FUNCTION_BLOCK FB_SerialCom
VAR_IN_OUT
	RxBuffer	: ComBuffer;
	TxBuffer	: ComBuffer;
END_VAR

VAR
	fbSend		: SendString;
	bSendBusy	: BOOL;
	eSendErrorID: ComError_t;
	bSend		: BOOL;
	bReceive		: BOOL := TRUE;
	sendsstriung: STRING;
	
	fbReceive:Receivestring;//接收功能宁符决块
	sedstring: STRING;
END_VAR
VAR_OUTPUT
	sReceivedString: STRING;//接收到的字符宏
END_VAR
VAR_IN_OUT
	// 發送出去的字串
	sSendString: STRING;
	sLastReceivedstring: STRING;//最后接收到的产符书
END_VAR
VAR
	bStringReceived : BOOL;
	bReceiveBusy: BOOL;
	breceiveError: BOOL;
	eReceiveErrorID : ComError_t;
	bReceiveTimeout: BOOL;
	nReceiveCounter: UDINT;
	sSendString_Len: int;
END_VAR

sedstring := CONCAT(STR1:= CONCAT(STR1:='$02' , STR2:= sSendString ), STR2:='$03' );
sSendString_Len := LEN (sSendString);
IF sSendString_Len > 0 OR fbSend.Busy THEN
	sSendString :='';
	sendsstriung:=sedstring;
	fbSend(
		SendString:=sedstring,
		TxBuffer:= 	TxBuffer,
		Busy=>bSendBusy,
		Error=>);
	IF fbSend.Error <> ComError_t.COMERROR_NOERROR THEN
		eSendErrorID := fbSend.Error;
	END_IF
END_IF
IF bReceive THEN	
	fbReceive(
		Prefix	:= '$02',
		Suffix	:= '$03',
		Timeout	:= T#1S,
		ReceivedString:=sReceivedString,
		RXbuffer := RxBuffer,
		StringReceived => bStringReceived,
		Busy => bReceiveBusy,
		Error=>,
		RxTimeout=>bReceiveTimeout);
	IF fbReceive.Error <> ComError_t.COMERROR_NOERROR THEN
			eReceiveErrorID := fbReceive.Error;
	END_IF

	IF bStringReceived THEN
		nReceiveCounter := nReceiveCounter + 1;
		sLastReceivedstring := sReceivedString;
	END_IF
END_IF

END_FUNCTION_BLOCK

(* stored: Version 1.1.0.1, ProductVersion 3.1.4024.10
   POU FB_SerialCom: Id {c70f9cc2-e962-4677-8a00-b9f8bf30f1ad}, SpecialFunc None *)
